FUNCTION TryConvert_DT_TO_BYTE : BOOL
VAR_INPUT
	in : DT;
	out : REFERENCE TO BYTE;
END_VAR

IF in > DatatypeLimits.MAX_VALUE_OF_DT_WHICH_CAN_BE_HELD_IN_A_BYTE THEN
	RETURN;
END_IF

out := DT_TO_BYTE(in);
TryConvert_DT_TO_BYTE := TRUE;

END_FUNCTION

(* stored: Version 1.1.0.1, ProductVersion 3.1.4024.12
   POU TryConvert_DT_TO_BYTE: Id {d1e4722a-dca6-4de5-829f-edaab6c049e8}, SpecialFunc None *)
